// TIA Portal V18 export
// export: Created 2026-06-08T17:01:58.7180031Z, ExportSetting WithDefaults, DisplayName Totally Integrated Automation Portal, DisplayVersion V18, DisplayName TIA Portal Openness, DisplayVersion V18, DisplayName TIA Portal Version Control Interface, DisplayVersion V18, DisplayName STEP 7 Professional, DisplayVersion V18, DisplayName STEP 7 Safety, DisplayVersion V18, DisplayName WinCC Professional, DisplayVersion V18
FUNCTION "M2_WIND_DOWN" : Void   // FC8, LAD
{ S7_Optimized_Access := 'TRUE' }
VERSION : 0.1
// stored: AutoNumber true, IsIECCheckEnabled false, SetENOAutomatically false, UDAEnableTagReadback false
BEGIN

REGION Network 1
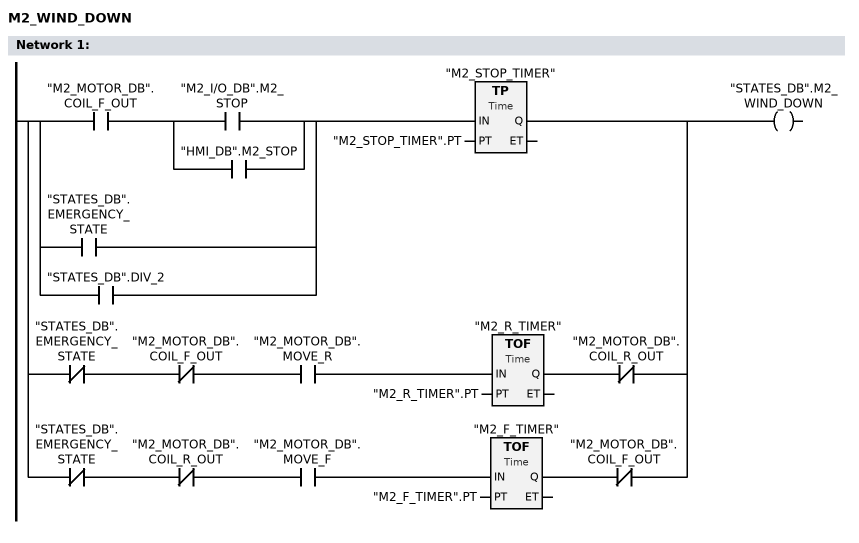
   RUNG wire#powerrail
      Contact( "M2_MOTOR_DB".COIL_F_OUT )
      wire#w1
      Contact( "M2_I/O_DB".M2_STOP )
      wire#w2
      { S7_Templates := "time_type := Time" } "M2_STOP_TIMER".TP(pt := "M2_STOP_TIMER".PT, et =>)
      wire#w3
      Coil( "STATES_DB".M2_WIND_DOWN )
   END_RUNG
   RUNG wire#w1
      Contact( "HMI_DB".M2_STOP )
   END_RUNG wire#w2
   RUNG wire#powerrail
      Contact( "STATES_DB".EMERGENCY_STATE )
   END_RUNG wire#w2
   RUNG wire#powerrail
      Contact( "STATES_DB".DIV_2 )
   END_RUNG wire#w2
   RUNG wire#powerrail
      I_Contact( "STATES_DB".EMERGENCY_STATE )
      I_Contact( "M2_MOTOR_DB".COIL_F_OUT )
      Contact( "M2_MOTOR_DB".MOVE_R )
      { S7_Templates := "time_type := Time" } "M2_R_TIMER".TOF(pt := "M2_R_TIMER".PT, et =>)
      I_Contact( "M2_MOTOR_DB".COIL_R_OUT )
   END_RUNG wire#w3
   RUNG wire#powerrail
      I_Contact( "STATES_DB".EMERGENCY_STATE )
      I_Contact( "M2_MOTOR_DB".COIL_R_OUT )
      Contact( "M2_MOTOR_DB".MOVE_F )
      { S7_Templates := "time_type := Time" } "M2_F_TIMER".TOF(pt := "M2_F_TIMER".PT, et =>)
      I_Contact( "M2_MOTOR_DB".COIL_F_OUT )
   END_RUNG wire#w3
   // the same network as SCL:
   "M2_STOP_TIMER".TP(IN := ("M2_MOTOR_DB".COIL_F_OUT AND ("M2_I/O_DB".M2_STOP OR "HMI_DB".M2_STOP)) OR "STATES_DB".EMERGENCY_STATE OR "STATES_DB".DIV_2,
                      PT := "M2_STOP_TIMER".PT);
   "M2_R_TIMER".TOF(IN := NOT "STATES_DB".EMERGENCY_STATE AND NOT "M2_MOTOR_DB".COIL_F_OUT AND "M2_MOTOR_DB".MOVE_R,
                    PT := "M2_R_TIMER".PT);
   "M2_F_TIMER".TOF(IN := NOT "STATES_DB".EMERGENCY_STATE AND NOT "M2_MOTOR_DB".COIL_R_OUT AND "M2_MOTOR_DB".MOVE_F,
                    PT := "M2_F_TIMER".PT);
   "STATES_DB".M2_WIND_DOWN := "M2_STOP_TIMER".Q OR ("M2_R_TIMER".Q AND NOT "M2_MOTOR_DB".COIL_R_OUT) OR ("M2_F_TIMER".Q AND NOT "M2_MOTOR_DB".COIL_F_OUT);
END_REGION
END_FUNCTION
